// TIA Portal project "Circuit to Ladder Logic Conversion Example" (V17)
// Siemens TIA Portal Tutorial: Circuit to Ladder Logic Conversion Example

(* hardware
DEVICE "S7-1200 station_1"  S7-1200 Station
   slot 0: "Rack_0"  S7-1200 Rack  Rack  V1.0
   slot 1: "PLC_1"  CPU 1211C AC/DC/Rly  6ES7 211-1BE40-0XB0  V4.5
*)

// ===== PLC "PLC_1"  CPU 1211C AC/DC/Rly =====

VAR_GLOBAL   // PLC tag table "Default tag table"
   "A" AT %I0.0 : Bool;
   "B" AT %I0.1 : Bool;
   "C" AT %I0.2 : Bool;
   "D" AT %I0.3 : Bool;
   "Y O/P" AT %Q0.0 : Bool;
END_VAR

ORGANIZATION_BLOCK "Main"   // OB1, LAD, ProgramCycle
TITLE = "Main Program Sweep (Cycle)"
{ S7_Optimized_Access := 'TRUE' }
VERSION : 0.1
   VAR_INPUT
      Initial_Call : Bool;   // Initial call of this OB
      Remanence : Bool;   // =True, if remanent data are available
   END_VAR
BEGIN

REGION Network 1
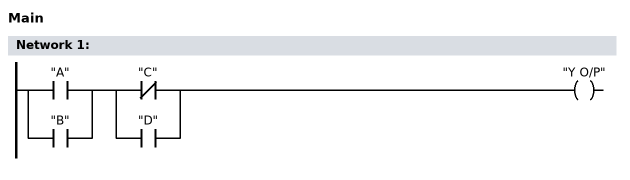
   RUNG wire#powerrail
      Contact( "A" )
      wire#w1
      I_Contact( "C" )
      wire#w2
      Coil( "Y O/P" )
   END_RUNG
   RUNG wire#powerrail
      Contact( "B" )
   END_RUNG wire#w1
   RUNG wire#w1
      Contact( "D" )
   END_RUNG wire#w2
   // the same network as SCL:
   "Y O/P" := ("A" OR "B") AND (NOT "C" OR "D");
END_REGION
END_ORGANIZATION_BLOCK